FUNCTION_BLOCK LinearMotionLoad (* Basic Function Block Type *)
  (* Standard: 61499-2 *)
  (* Version 0.0, 12/5/2011, XPMUser, nxtControl GmbH, Template *)
  PACKAGE Main;
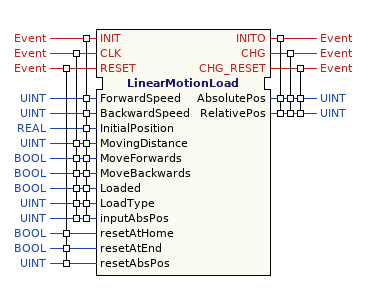
  EVENT_INPUT
    INIT WITH ForwardSpeed, BackwardSpeed, InitialPosition, MovingDistance, MoveForwards, MoveBackwards, Loaded, LoadType, inputAbsPos; (* Initialization Request *)
    CLK WITH MovingDistance, MoveForwards, MoveBackwards, Loaded, LoadType, inputAbsPos; (* Clock signal *)
    RESET WITH resetAtHome, resetAtEnd, resetAbsPos;
  END_EVENT
  EVENT_OUTPUT
    INITO WITH RelativePos, AbsolutePos; (* Initialization Confirm *)
    CHG WITH RelativePos, AbsolutePos; (* Indicates changes on the data output *)
    CHG_RESET WITH AbsolutePos, RelativePos;
  END_EVENT
  VAR_INPUT
    ForwardSpeed : UINT; (* Forward speed *)
    BackwardSpeed : UINT; (* Backward speed *)
    InitialPosition : REAL; (* Absolute initial position *)
    MovingDistance : UINT;
    MoveForwards : BOOL; (* Move forwards *)
    MoveBackwards : BOOL; (* Move backwards *)
    Loaded : BOOL;
    LoadType : UINT; (* With different types of load, the actual moving speed varies *)
    inputAbsPos : UINT;
    resetAtHome : BOOL;
    resetAtEnd : BOOL;
    resetAbsPos : UINT;
  END_VAR
  VAR_OUTPUT
    AbsolutePos : UINT;
    RelativePos : UINT; (* Position in percentation *)
  END_VAR
  VAR
    percentagePos : REAL;
  END_VAR
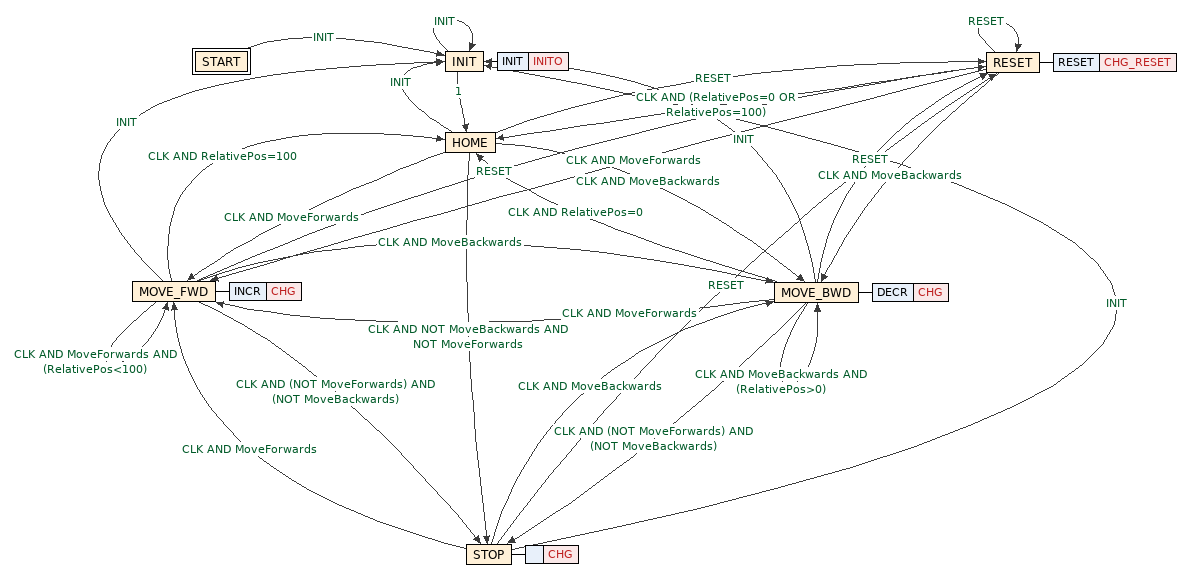
  EC_STATES
    START; (* Initial State *)
    INIT : INIT -> INITO; (* Initialization *)
    MOVE_FWD : INCR -> CHG;
    MOVE_BWD : DECR -> CHG;
    STOP : -> CHG;
    HOME; (* At home position *)
    RESET : RESET -> CHG_RESET;
  END_STATES
  EC_TRANSITIONS
    START TO INIT := INIT;
    INIT TO HOME := 1;
    HOME TO MOVE_FWD := CLK AND MoveForwards;
    MOVE_FWD TO STOP := CLK AND (NOT MoveForwards) AND (NOT MoveBackwards);
    MOVE_BWD TO STOP := CLK AND (NOT MoveForwards) AND (NOT MoveBackwards);
    STOP TO MOVE_FWD := CLK AND MoveForwards;
    STOP TO MOVE_BWD := CLK AND MoveBackwards;
    MOVE_BWD TO HOME := CLK AND RelativePos=0;
    MOVE_FWD TO MOVE_BWD := CLK AND MoveBackwards;
    MOVE_BWD TO MOVE_FWD := CLK AND MoveForwards;
    MOVE_FWD TO MOVE_FWD := CLK AND MoveForwards AND (RelativePos<100);
    MOVE_BWD TO MOVE_BWD := CLK AND MoveBackwards AND (RelativePos>0);
    HOME TO MOVE_BWD := CLK AND MoveBackwards;
    MOVE_FWD TO HOME := CLK AND RelativePos=100;
    HOME TO INIT := INIT;
    MOVE_BWD TO INIT := INIT;
    MOVE_FWD TO INIT := INIT;
    STOP TO INIT := INIT;
    INIT TO INIT := INIT;
    HOME TO RESET := RESET;
    MOVE_BWD TO RESET := RESET;
    MOVE_FWD TO RESET := RESET;
    RESET TO MOVE_BWD := CLK AND MoveBackwards;
    RESET TO MOVE_FWD := CLK AND MoveForwards;
    RESET TO HOME := CLK AND (RelativePos=0 OR RelativePos=100);
    RESET TO RESET := RESET;
    HOME TO STOP := CLK AND NOT MoveBackwards AND NOT MoveForwards;
    STOP TO RESET := RESET;
  END_TRANSITIONS
  ALGORITHM INIT IN ST: (* Initialization algorithm *)
INIT:=FALSE;
AbsolutePos := REAL_TO_UINT(InitialPosition);
AbsolutePos := inputAbsPos + AbsolutePos;
RelativePos := 0;
percentagePos := 0;
  END_ALGORITHM
  ALGORITHM INCR IN ST: (* Increment the position *)
VAR
    position: REAL;
END_VAR
(* ---------- Check whether the motor is loaded ----------*)
CLK := FALSE;
IF (Loaded AND LoadType > 0) THEN
    position := (AbsolutePos + ForwardSpeed * ((1 - LoadType) / 10));
    IF (position > MovingDistance) THEN
        position := MovingDistance;
    END_IF;
    percentagePos := (position / MovingDistance) * 100;
ELSE
    position := AbsolutePos + ForwardSpeed;
    IF (position > MovingDistance) THEN
        position := MovingDistance;
    END_IF;
    percentagePos := (position / MovingDistance) * 100;
END_IF;
AbsolutePos := REAL_TO_UINT(position);
AbsolutePos := inputAbsPos + AbsolutePos;
RelativePos := REAL_TO_UINT(percentagePos);
  END_ALGORITHM
  ALGORITHM DECR IN ST: (* Decrement the position *)
VAR
    position: REAL;
END_VAR
(* ---------- Check whether the motor is loaded ----------*)
CLK := FALSE;
IF (Loaded AND LoadType > 0) THEN
    position := (AbsolutePos - BackwardSpeed * (1 - LoadType / 10));
    IF (AbsolutePos > 0) THEN
        position := AbsolutePos - BackwardSpeed;
    ELSE
        position := 0;
    END_IF;
    percentagePos := (position / MovingDistance) * 100;
ELSE
    IF (AbsolutePos > 0) THEN
        position := AbsolutePos - BackwardSpeed;
   ELSE
        position := 0;
    END_IF;
    percentagePos := (position / MovingDistance) * 100;
END_IF;
AbsolutePos := REAL_TO_UINT(position);
RelativePos := REAL_TO_UINT(percentagePos);
  END_ALGORITHM
  ALGORITHM RESET IN ST:
RESET:=FALSE;
IF (resetAtEnd=TRUE AND resetAtHome=FALSE) THEN
	AbsolutePos := inputAbsPos + 100;
ELSIF (resetAtEnd=FALSE AND resetAtHome=TRUE) THEN
	AbsolutePos := inputAbsPos;
ELSIF (resetAtEnd=FALSE AND resetAtHome=FALSE) THEN
	AbsolutePos := resetAbsPos;
END_IF;
IF (AbsolutePos > MovingDistance) THEN
  AbsolutePos := MovingDistance;
END_IF;
RelativePos := (AbsolutePos / MovingDistance) * 100;
  END_ALGORITHM
END_FUNCTION_BLOCK
